(* PLC project Desconhecido, UFSCar Conversor PNML2Ladder 1 *)
(* stored: creationDateTime 2025-01-15T12:13:14, modificationDateTime 2025-02-12T15:17:24 *)

PROGRAM instance0

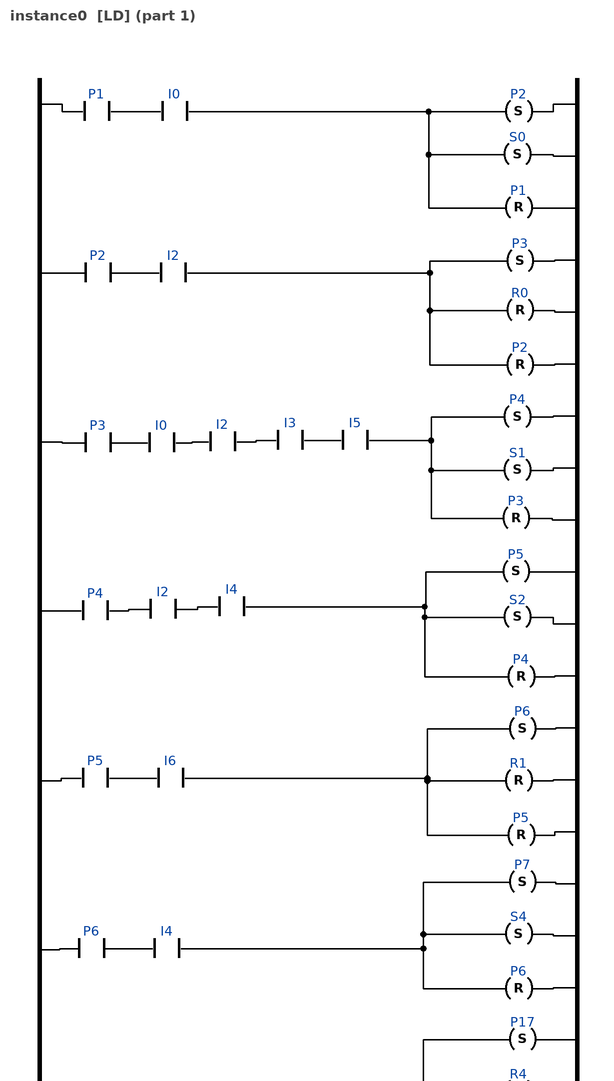
(* LD diagram, written out as Structured Text *)
IF P1 AND I0 THEN P2 := TRUE; END_IF;
IF P1 AND I0 THEN S0 := TRUE; END_IF;
IF P1 AND I0 THEN P1 := FALSE; END_IF;
IF P2 AND I2 THEN P3 := TRUE; END_IF;
IF P2 AND I2 THEN R0 := FALSE; END_IF;
IF P2 AND I2 THEN P2 := FALSE; END_IF;
IF P3 AND I0 AND I2 AND I3 AND I5 THEN P3 := FALSE; END_IF;
IF P3 AND I0 AND I2 AND I3 AND I5 THEN P4 := TRUE; END_IF;
IF P3 AND I0 AND I2 AND I3 AND I5 THEN S1 := TRUE; END_IF;
IF P4 AND I2 AND I4 THEN P5 := TRUE; END_IF;
IF P4 AND I2 AND I4 THEN S2 := TRUE; END_IF;
IF P4 AND I2 AND I4 THEN P4 := FALSE; END_IF;
IF P5 AND I6 THEN P6 := TRUE; END_IF;
IF P5 AND I6 THEN R1 := FALSE; END_IF;
IF P5 AND I6 THEN P5 := FALSE; END_IF;
IF P6 AND I4 THEN P7 := TRUE; END_IF;
IF P6 AND I4 THEN S4 := TRUE; END_IF;
IF P6 AND I4 THEN P6 := FALSE; END_IF;
IF P7 AND I8 THEN P17 := TRUE; END_IF;
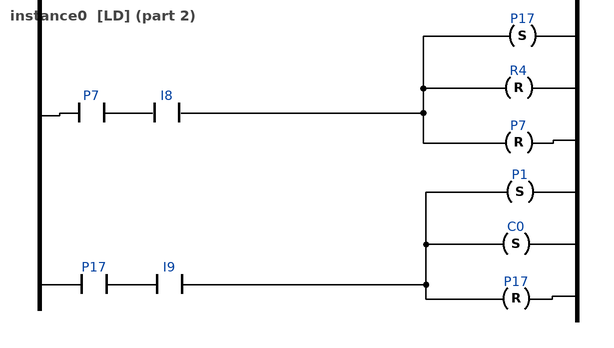
IF P7 AND I8 THEN R4 := FALSE; END_IF;
IF P7 AND I8 THEN P7 := FALSE; END_IF;
IF P17 AND I9 THEN P1 := TRUE; END_IF;
IF P17 AND I9 THEN C0 := TRUE; END_IF;
IF P17 AND I9 THEN P17 := FALSE; END_IF;
END_PROGRAM

CONFIGURATION config0
  RESOURCE resource1 ON PLC
    TASK task0(INTERVAL := T#20ms, PRIORITY := 0);
    PROGRAM instance0 WITH task0 : program0;
  END_RESOURCE
END_CONFIGURATION
